// TIA Portal V17 export
// export: Created 2022-07-28T18:02:45.188659Z, ExportSetting None, DisplayName Totally Integrated Automation Portal, DisplayVersion V17, DisplayName TIA Portal Openness, DisplayVersion V17, DisplayName TIA Portal Teamcenter Gateway, DisplayVersion V17, DisplayName TIA Portal Version Control Interface, DisplayVersion V17, DisplayName TIA Portal Test Suite Advanced, DisplayVersion V17, DisplayName SINAMICS Startdrive Advanced, DisplayVersion V17, DisplayName SINAMICS DCC, DisplayVersion V17, DisplayName SINAMICS Startdrive G130, G150, S120, S150, SINAMICS MV, S210, DisplayVersion V17, DisplayName SINAMICS Startdrive G110M, G120, G120C, G120D, G120P, G115D, DisplayVersion V17, DisplayName STEP 7 Professional, DisplayVersion V17, DisplayName SIMATIC Energy Suite, DisplayVersion V17, DisplayName STEP 7 CFC, DisplayVersion V17, DisplayName STEP 7 Safety, DisplayVersion V17, DisplayName WinCC Advanced / Unified PC, DisplayVersion V17, DisplayName SIMATIC Visualization Architect, DisplayVersion V17
FUNCTION "Lib_FC_DSens_CycleInfo_Count_State" : Void   // FC9, SCL
{ S7_Optimized_Access := 'TRUE' }
// stored: SetENOAutomatically false
   VAR_INPUT
      Alarm : Bool;
      AlarmNew : Bool;
      Warning : Bool;
      WarningNew : Bool;
      Simulation : Bool;
   END_VAR
   VAR_IN_OUT
      PLC_CycleInfo : "Lib_PLC_CycleInfo";
   END_VAR
BEGIN


   REGION PLC State + Counter  
       //----------------------------------------------
       IF #Alarm THEN
           #PLC_CycleInfo.Alarm.Alarm := TRUE;//  =1, є хоча б одна    
           #PLC_CycleInfo.Counter.Alarm := #PLC_CycleInfo.Counter.Alarm + 1;
       END_IF;
       IF #Warning THEN
           #PLC_CycleInfo.Alarm.Warning := TRUE;//  =1, є хоча б одна  
           #PLC_CycleInfo.Counter.Warning := #PLC_CycleInfo.Counter.Warning + 1;
       END_IF;
       IF #Simulation THEN
           #PLC_CycleInfo.State.Simulation := TRUE;
       END_IF;


       IF #AlarmNew THEN
           #PLC_CycleInfo.Alarm.AlarmNew := true;
       END_IF;
       IF #WarningNew THEN
           #PLC_CycleInfo.Alarm.WarningNew := true;
       END_IF;
       //----------------------------------------------
   END_REGION
END_FUNCTION
